_CFC_ (* Continuous Function Chart, elements in execution order *)
#0 RS_UST_BLOK:R_TRIG(CLK: SHU6_PV1_UST_RE_RABOTA)
#1 RS_SB_BLOK:R_TRIG(CLK: NOT SHU6_PV1_UST_RE_RABOTA)
#2 RS_BLOKIROVKA:RS(SET: #0.Q, RESET1: #1.Q)
#3 SHU6_PV1_BLOK_YA3 <= #2.Q1
#4 SHU6_PV1_BLOK_RQ1 <= NOT #2.Q1
#5 SHU6_PV1_BLOK_YA4 <= #2.Q1
#6 MUL(SHU6_PV1_RQ1_MAX_RAB_CH, 0.95)
#7 res_1 <= #6
#8 >(#6, SHU6_RQ1_REQ_VYHOD)
#9 res_2 <= #8
#10 >(SHU6_YA3_REQ_VYHOD, 5)
#11 >(SHU6_YA4_REQ_VYHOD, 5)
#12 OR(#10, #11)
#13 AND(res_2, #12)
#14 SHU6_PV1_BLOK_YA3 <= NOT #13
#15 SHU6_PV1_BLOK_RQ1 <= #13
#16 SHU6_PV1_BLOK_YA4 <= NOT #13
#17 <(SHU6_YA3_REQ_VYHOD, 5)
#18 AND(SHU6_PV1_UST_RE_RABOTA, #17)
#19 <(SHU6_RQ1_REQ_VYHOD, res_1)
#20 AND(#18, #19)
#21 SHU6_PV1_BLOK_YA3 <= #20
#22 SHU6_PV1_BLOK_RQ1 <= NOT #20
#23 <(SHU6_YA4_REQ_VYHOD, 5)
#24 AND(SHU6_PV1_UST_RE_RABOTA, #23)
#25 <(SHU6_RQ1_REQ_VYHOD, res_1)
#26 AND(#24, #25)
#27 SHU6_PV1_BLOK_YA4 <= #26
#28 SHU6_PV1_BLOK_RQ1 <= NOT #26
#29 SEL(SHU6_PV1_BLOK_RQ1, SHU6_RQ1_REQ_VYHOD, res_1)
#30 MOVE(#29)
#31 SHU6_RQ1_SPEEDMOTOR <= #30
#32 SEL(SHU6_PV1_YARQ1_DI6_M, #29, SHU6_PV1_MRQ1_ZAD_RUCH)
#33 SHU6_PV1_RQ1_ZAD_VN <= #32
#34 OR(SHU6_PV1_BLOK_YA4, SHU6_PV1_UST_ZIMA)
#35 AND(#34, YA4_AVT)
#36 SEL(#35, SHU6_YA4_REQ_VYHOD, 0)
#37 SHU6_PV1_YA4_ZAD_VN <= #36
#38 OR(SHU6_PV1_BLOK_YA3, SHU6_PV1_UST_LETO)
#39 AND(NOT Z_ZAM_SR, YA3_AVT)
#40 AND(#38, #39)
#41 SEL(#40, SHU6_YA3_REQ_VYHOD, 0)
#42 SHU6_PV1_YA3_ZAD_VN <= #41
_END_CFC_
END_PROGRAM

(* POU Output/ALL_Output, CFC *)
PROGRAM ALL_Output
VAR
END_VAR
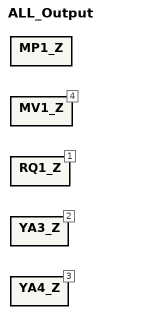
_CFC_ (* Continuous Function Chart, elements in execution order *)
#0 MP1_Z()
#1 RQ1_Z()
#2 YA3_Z()
#3 YA4_Z()
#4 MV1_Z()
_END_CFC_
(* the same logic as Structured Text *)
MP1_Z();
RQ1_Z();
YA3_Z();
YA4_Z();
MV1_Z();
END_PROGRAM

(* POU Output/AO/MP1_Z, CFC *)
PROGRAM MP1_Z
VAR
	fb_HVACAO_SHU6_PV1_UZ1_AO1: FB_HVACAnalogOutput;
	enableFeedbCtrl: BOOL := FALSE;
	hysFbCtrl: REAL := 0;
	direction: BOOL;
	delay: TIME := T#0s;
	hi: REAL := 50;
	low: REAL := 0;

END_VAR
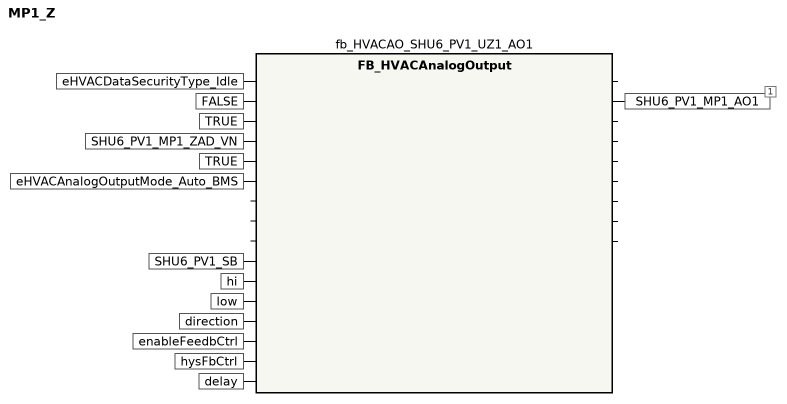
_CFC_ (* Continuous Function Chart, elements in execution order *)
#0 fb_HVACAO_SHU6_PV1_UZ1_AO1:FB_HVACAnalogOutput(eHVACDataSecurityType_Idle, FALSE, TRUE, SHU6_PV1_MP1_ZAD_VN, TRUE, eHVACAnalogOutputMode_Auto_BMS, -, -, -, SHU6_PV1_SB, hi, low, direction, enableFeedbCtrl, hysFbCtrl, delay)
#1 SHU6_PV1_MP1_AO1 <= #0.out 2
_END_CFC_
END_PROGRAM

(* POU Output/AO/RQ1_Z, CFC *)
PROGRAM RQ1_Z
VAR
	fb_HVACAO_SHU6_PV1_RQ1_AO5: FB_HVACAnalogOutput;
         enableFeedbCtrl: BOOL := FALSE;
         hysFbCtrl: REAL := 0;
        direction: BOOL;
        delay: TIME := T#0s;
        hi: REAL := 50;
        low: REAL := 0;
END_VAR
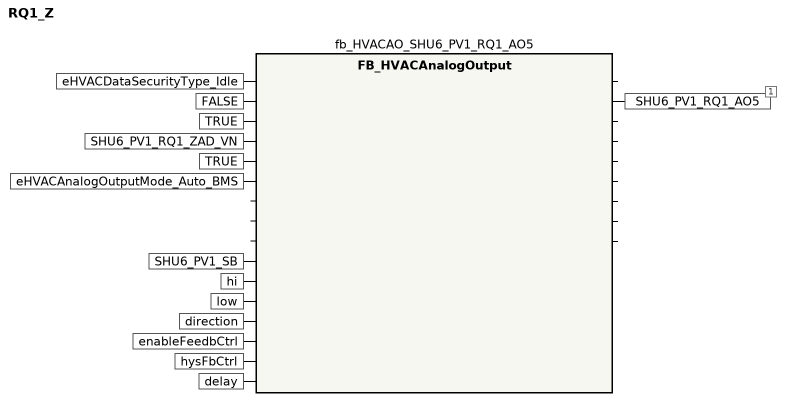
_CFC_ (* Continuous Function Chart, elements in execution order *)
#0 fb_HVACAO_SHU6_PV1_RQ1_AO5:FB_HVACAnalogOutput(eHVACDataSecurityType_Idle, FALSE, TRUE, SHU6_PV1_RQ1_ZAD_VN, TRUE, eHVACAnalogOutputMode_Auto_BMS, -, -, -, SHU6_PV1_SB, hi, low, direction, enableFeedbCtrl, hysFbCtrl, delay)
#1 SHU6_PV1_RQ1_AO5 <= #0.out 2
_END_CFC_
END_PROGRAM

(* POU Output/AO/YA3_Z, CFC *)
PROGRAM YA3_Z
VAR
	fb_HVACAO_SHU6_PV1_PV1_AO6: FB_HVACAnalogOutput;
	enableFeedbCtrl: BOOL := FALSE;
	hysFbCtrl: REAL := 0;
	direction: BOOL;
	delay: TIME := T#0s;
END_VAR
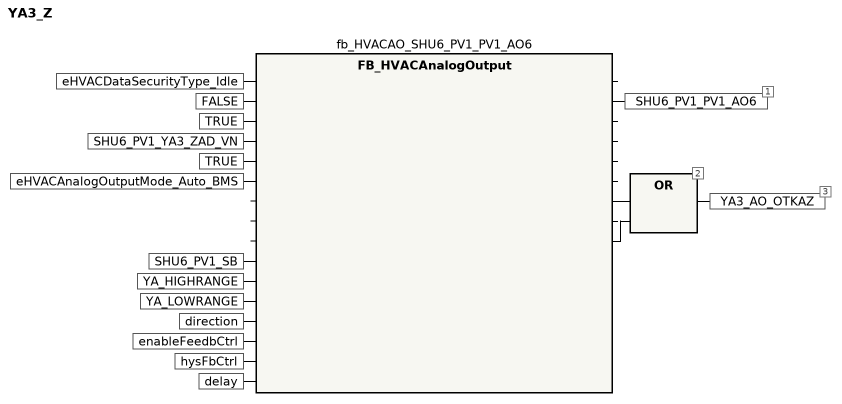
_CFC_ (* Continuous Function Chart, elements in execution order *)
#0 fb_HVACAO_SHU6_PV1_PV1_AO6:FB_HVACAnalogOutput(eHVACDataSecurityType_Idle, FALSE, TRUE, SHU6_PV1_YA3_ZAD_VN, TRUE, eHVACAnalogOutputMode_Auto_BMS, -, -, -, SHU6_PV1_SB, YA_HIGHRANGE, YA_LOWRANGE, direction, enableFeedbCtrl, hysFbCtrl, delay)
#1 SHU6_PV1_PV1_AO6 <= #0.out 2
#2 OR(#0.out 7, #0.out 9)
#3 YA3_AO_OTKAZ <= #2
_END_CFC_
END_PROGRAM

(* POU Output/AO/YA4_Z, CFC *)
PROGRAM YA4_Z
VAR
	fb_HVACAO_SHU6_PV1_PV1_AO7: FB_HVACAnalogOutput;
	enableFeedbCtrl: BOOL := FALSE;
	hysFbCtrl: REAL := 0;
	direction: BOOL;
	delay: TIME := T#0s;
END_VAR
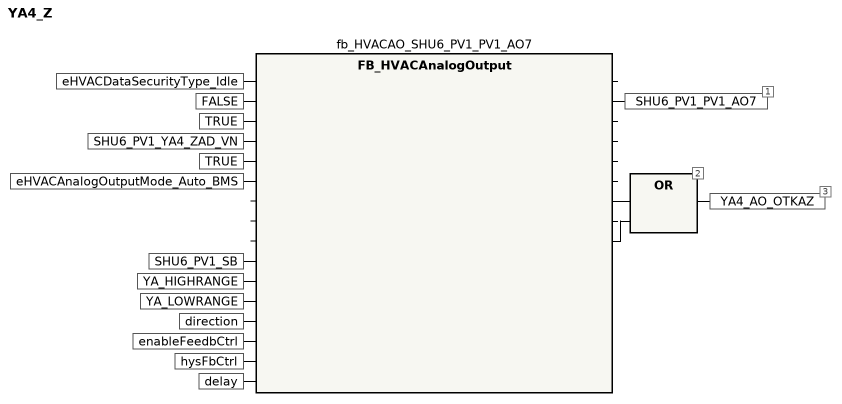
_CFC_ (* Continuous Function Chart, elements in execution order *)
#0 fb_HVACAO_SHU6_PV1_PV1_AO7:FB_HVACAnalogOutput(eHVACDataSecurityType_Idle, FALSE, TRUE, SHU6_PV1_YA4_ZAD_VN, TRUE, eHVACAnalogOutputMode_Auto_BMS, -, -, -, SHU6_PV1_SB, YA_HIGHRANGE, YA_LOWRANGE, direction, enableFeedbCtrl, hysFbCtrl, delay)
#1 SHU6_PV1_PV1_AO7 <= #0.out 2
#2 OR(#0.out 7, #0.out 9)
#3 YA4_AO_OTKAZ <= #2
_END_CFC_
END_PROGRAM

(* POU Output/AO/MV1_Z, CFC *)
PROGRAM MV1_Z
VAR
	enableFeedbCtrl: BOOL := FALSE;
	hysFbCtrl: REAL := 0;
	direction: BOOL;
	delay: TIME := T#0s;
	hi: REAL := 50;
	low: REAL := 0;
	fb_HVACAO_SHU6_PV1_UZ3_AO2: FB_HVACAnalogOutput;
END_VAR
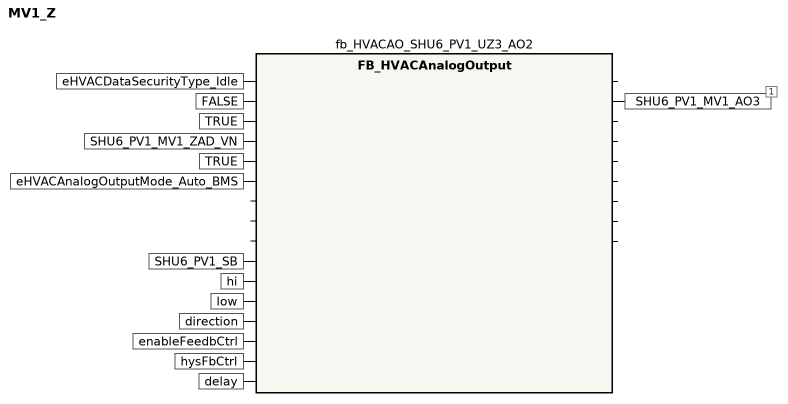
_CFC_ (* Continuous Function Chart, elements in execution order *)
#0 fb_HVACAO_SHU6_PV1_UZ3_AO2:FB_HVACAnalogOutput(eHVACDataSecurityType_Idle, FALSE, TRUE, SHU6_PV1_MV1_ZAD_VN, TRUE, eHVACAnalogOutputMode_Auto_BMS, -, -, -, SHU6_PV1_SB, hi, low, direction, enableFeedbCtrl, hysFbCtrl, delay)
#1 SHU6_PV1_MV1_AO3 <= #0.out 2
_END_CFC_
END_PROGRAM

(* POU Input/CI/ModBus_M, CFC *)
PROGRAM ModBus_M
VAR
	MB_READ_REGS: ModbusRtuMaster_KL6x22B;
	Quantity: WORD:= 4;
	MBAddr: WORD:= 16#3000;

	CTU_ModBus: CTU;
	TON1: TON;
	TON2: TON;


	RT_ModBus: R_TRIG;

	Errorld: MODBUS_ERRORS;
	cbRead: UINT;
	TOF1: TOF;
END_VAR
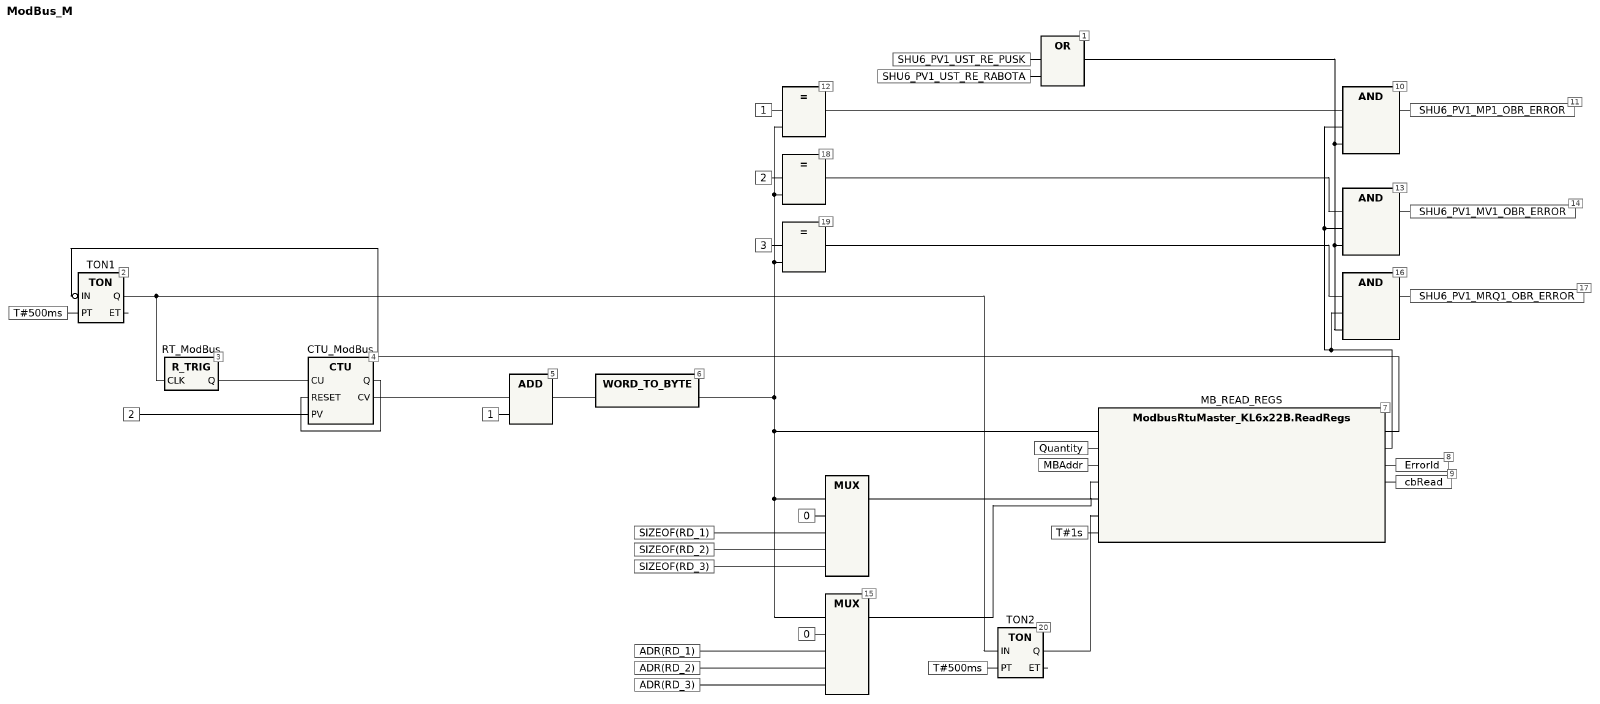
